// TIA Portal V19 export
FUNCTION_BLOCK "Main_Safety_RTG1"   // FB1, F_LAD
{ S7_Optimized_Access := 'TRUE' }
// stored: AutoNumber false
   VAR_TEMP
      EstopLamp : Bool;
   END_VAR
   VAR_TEMP   // added for the SCL form of the ladder/FBD networks
      _w1 : Bool;
   END_VAR
BEGIN

REGION Network 1
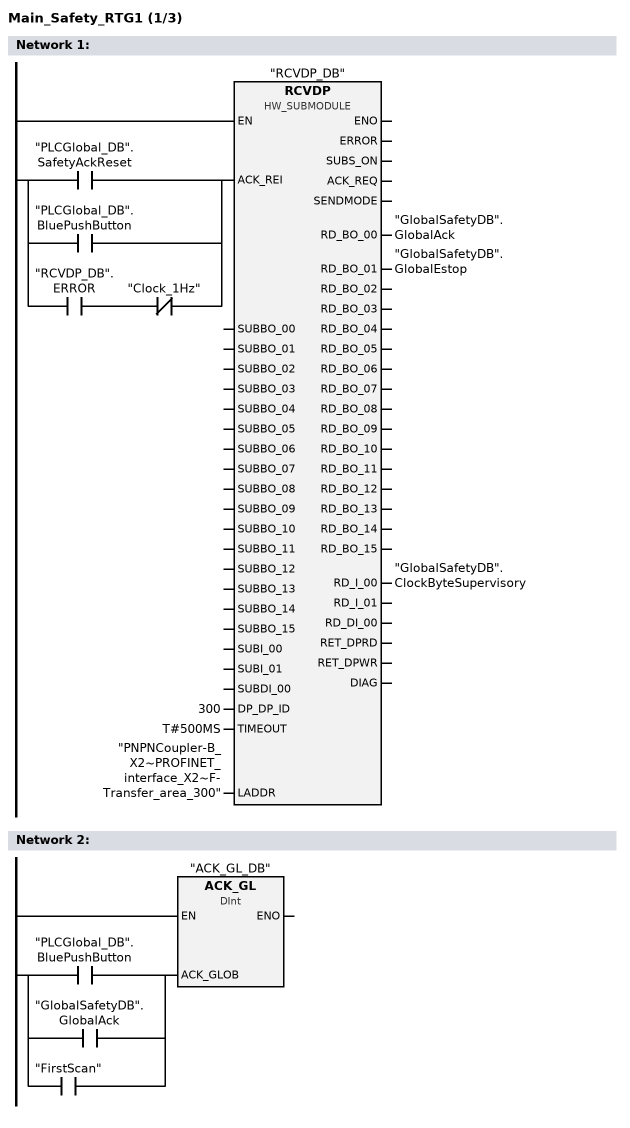
   RUNG wire#powerrail
      { S7_Templates := "laddr_type := HW_SUBMODULE" } "RCVDP_DB".RCVDP(ACK_REI := wire#w1, SUBBO_00 :=, SUBBO_01 :=, SUBBO_02 :=, SUBBO_03 :=, SUBBO_04 :=, SUBBO_05 :=, SUBBO_06 :=, SUBBO_07 :=, SUBBO_08 :=, SUBBO_09 :=, SUBBO_10 :=, SUBBO_11 :=, SUBBO_12 :=, SUBBO_13 :=, SUBBO_14 :=, SUBBO_15 :=, SUBI_00 :=, SUBI_01 :=, SUBDI_00 :=, DP_DP_ID := 300, TIMEOUT := T#500MS, LADDR := "PNPNCoupler-B_X2~PROFINET_interface_X2~F-Transfer_area_300", ERROR =>, SUBS_ON =>, ACK_REQ =>, SENDMODE =>, RD_BO_00 => "GlobalSafetyDB".GlobalAck, RD_BO_01 => "GlobalSafetyDB".GlobalEstop, RD_BO_02 =>, RD_BO_03 =>, RD_BO_04 =>, RD_BO_05 =>, RD_BO_06 =>, RD_BO_07 =>, RD_BO_08 =>, RD_BO_09 =>, RD_BO_10 =>, RD_BO_11 =>, RD_BO_12 =>, RD_BO_13 =>, RD_BO_14 =>, RD_BO_15 =>, RD_I_00 => "GlobalSafetyDB".ClockByteSupervisory, RD_I_01 =>, RD_DI_00 =>, RET_DPRD =>, RET_DPWR =>, DIAG =>)
   END_RUNG
   RUNG wire#powerrail
      Contact( "PLCGlobal_DB".SafetyAckReset )
   END_RUNG wire#w1
   RUNG wire#powerrail
      Contact( "PLCGlobal_DB".BluePushButton )
   END_RUNG wire#w1
   RUNG wire#powerrail
      Contact( "RCVDP_DB".ERROR )
      I_Contact( "Clock_1Hz" )
   END_RUNG wire#w1
   // the same network as SCL:
   "RCVDP_DB"(ACK_REI := "PLCGlobal_DB".SafetyAckReset OR "PLCGlobal_DB".BluePushButton OR ("RCVDP_DB".ERROR AND NOT "Clock_1Hz"),   // RCVDP
              DP_DP_ID := 300,
              TIMEOUT := T#500MS,
              LADDR := "PNPNCoupler-B_X2~PROFINET_interface_X2~F-Transfer_area_300",
              RD_BO_00 => "GlobalSafetyDB".GlobalAck,
              RD_BO_01 => "GlobalSafetyDB".GlobalEstop,
              RD_I_00 => "GlobalSafetyDB".ClockByteSupervisory);
END_REGION

REGION Network 2
   RUNG wire#powerrail
      { S7_Templates := "codedbool_type := DInt" } "ACK_GL_DB".ACK_GL(ACK_GLOB := wire#w1)
   END_RUNG
   RUNG wire#powerrail
      Contact( "PLCGlobal_DB".BluePushButton )
   END_RUNG wire#w1
   RUNG wire#powerrail
      Contact( "GlobalSafetyDB".GlobalAck )
   END_RUNG wire#w1
   RUNG wire#powerrail
      Contact( "FirstScan" )
   END_RUNG wire#w1
   // the same network as SCL:
   "ACK_GL_DB"(ACK_GLOB := "PLCGlobal_DB".BluePushButton OR "GlobalSafetyDB".GlobalAck OR "FirstScan");   // ACK_GL
END_REGION

REGION Network 3
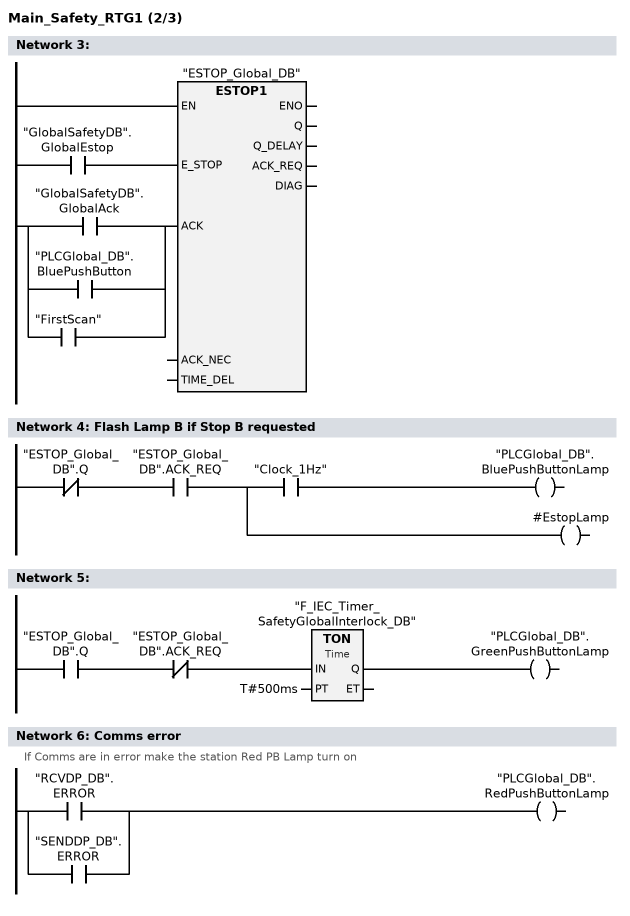
   RUNG wire#powerrail
      "ESTOP_Global_DB".ESTOP1(E_STOP := wire#w1, ACK := wire#w2, ACK_NEC :=, TIME_DEL :=, Q =>, Q_DELAY =>, ACK_REQ =>, DIAG =>)
   END_RUNG
   RUNG wire#powerrail
      Contact( "GlobalSafetyDB".GlobalEstop )
   END_RUNG wire#w1
   RUNG wire#powerrail
      Contact( "GlobalSafetyDB".GlobalAck )
   END_RUNG wire#w2
   RUNG wire#powerrail
      Contact( "PLCGlobal_DB".BluePushButton )
   END_RUNG wire#w2
   RUNG wire#powerrail
      Contact( "FirstScan" )
   END_RUNG wire#w2
   // the same network as SCL:
   "ESTOP_Global_DB"(E_STOP := "GlobalSafetyDB".GlobalEstop,   // ESTOP1
                     ACK := "GlobalSafetyDB".GlobalAck OR "PLCGlobal_DB".BluePushButton OR "FirstScan");
END_REGION

REGION Network 4: Flash Lamp B if Stop B requested
   RUNG wire#powerrail
      I_Contact( "ESTOP_Global_DB".Q )
      Contact( "ESTOP_Global_DB".ACK_REQ )
      wire#w1
      Contact( "Clock_1Hz" )
      Coil( "PLCGlobal_DB".BluePushButtonLamp )
   END_RUNG
   RUNG wire#w1
      Coil( #EstopLamp )
   END_RUNG
   // the same network as SCL:
   #_w1 := NOT "ESTOP_Global_DB".Q AND "ESTOP_Global_DB".ACK_REQ;
   "PLCGlobal_DB".BluePushButtonLamp := #_w1 AND "Clock_1Hz";
   #EstopLamp := #_w1;
END_REGION

REGION Network 5
   RUNG wire#powerrail
      Contact( "ESTOP_Global_DB".Q )
      I_Contact( "ESTOP_Global_DB".ACK_REQ )
      { S7_Templates := "[time_type := Time, codedbool_type := DInt]" } "F_IEC_Timer_SafetyGlobalInterlock_DB".TON(pt := T#500ms, et =>)
      Coil( "PLCGlobal_DB".GreenPushButtonLamp )
   END_RUNG
   // the same network as SCL:
   "F_IEC_Timer_SafetyGlobalInterlock_DB".TON(IN := "ESTOP_Global_DB".Q AND NOT "ESTOP_Global_DB".ACK_REQ,
                           PT := T#500ms);
   "PLCGlobal_DB".GreenPushButtonLamp := "F_IEC_Timer_SafetyGlobalInterlock_DB".Q;
END_REGION

REGION Network 6: Comms error
   // If Comms are in error make the station Red PB Lamp turn on
   RUNG wire#powerrail
      Contact( "RCVDP_DB".ERROR )
      wire#w1
      Coil( "PLCGlobal_DB".RedPushButtonLamp )
   END_RUNG
   RUNG wire#powerrail
      Contact( "SENDDP_DB".ERROR )
   END_RUNG wire#w1
   // the same network as SCL:
   "PLCGlobal_DB".RedPushButtonLamp := "RCVDP_DB".ERROR OR "SENDDP_DB".ERROR;
END_REGION

REGION Network 7
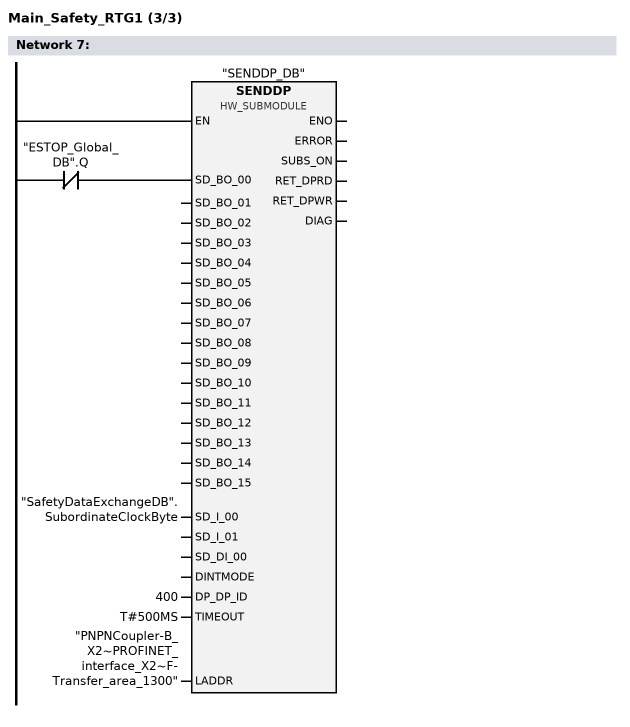
   RUNG wire#powerrail
      { S7_Templates := "laddr_type := HW_SUBMODULE" } "SENDDP_DB".SENDDP(SD_BO_00 := wire#w1, SD_BO_01 :=, SD_BO_02 :=, SD_BO_03 :=, SD_BO_04 :=, SD_BO_05 :=, SD_BO_06 :=, SD_BO_07 :=, SD_BO_08 :=, SD_BO_09 :=, SD_BO_10 :=, SD_BO_11 :=, SD_BO_12 :=, SD_BO_13 :=, SD_BO_14 :=, SD_BO_15 :=, SD_I_00 := "SafetyDataExchangeDB".SubordinateClockByte, SD_I_01 :=, SD_DI_00 :=, DINTMODE :=, DP_DP_ID := 400, TIMEOUT := T#500MS, LADDR := "PNPNCoupler-B_X2~PROFINET_interface_X2~F-Transfer_area_1300", ERROR =>, SUBS_ON =>, RET_DPRD =>, RET_DPWR =>, DIAG =>)
   END_RUNG
   RUNG wire#powerrail
      I_Contact( "ESTOP_Global_DB".Q )
   END_RUNG wire#w1
   // the same network as SCL:
   "SENDDP_DB"(SD_BO_00 := NOT "ESTOP_Global_DB".Q,   // SENDDP
               SD_I_00 := "SafetyDataExchangeDB".SubordinateClockByte,
               DP_DP_ID := 400,
               TIMEOUT := T#500MS,
               LADDR := "PNPNCoupler-B_X2~PROFINET_interface_X2~F-Transfer_area_1300");
END_REGION
END_FUNCTION_BLOCK
